// TIA Portal V16 export
// export: Created 2021-04-11T09:51:30.5050316Z, ExportSetting WithDefaults, DisplayName Totally Integrated Automation Portal, DisplayVersion V16, DisplayName TIA Portal Version Control Interface, DisplayVersion V16, DisplayName TIA Portal Openness, DisplayVersion V16, DisplayName STEP 7 Professional, DisplayVersion V16, DisplayName STEP 7 Safety, DisplayVersion V16, DisplayName WinCC Unified SCADA Engineering System, DisplayVersion V16
TYPE "recipeVar"
// stored: IsFailsafeCompliant false
   STRUCT
      setWeight : Real;   // весовая уставка в рецепте
      speed_InConveyer : Int;   // скорость конвейера питателя( конвейер на входе системы)
      speedVibro : Int;   // скорость вибролотков(одна на все)
      maxWeightBunker : Real;   // максимальный вес бункеров
      workPlavnik : Bool;   // работа плавника
      measurmentError : Real;   // допускаемая погрешность веса в общем сбросе
      mediumWeightProduct : Real;   // средний вес продукта
   END_STRUCT;
END_TYPE
